// TwinCAT 3 PLC project PLC_Classification
// ProgramVersion: 3.1.4024.0
// libraries:
//   Tc2_Standard, * (Beckhoff Automation GmbH)
//   Tc2_System, * (Beckhoff Automation GmbH)
//   Tc3_Module, * (Beckhoff Automation GmbH)
//   Tc3_Vision, * (Beckhoff Automation GmbH)
// project tree:
//   DUTs/ ST_ClassifierParams.TcDUT, E_ClassifierType.TcDUT, ESvmClassifierType.TcDUT
//   / PlcTask.TcTTO
//   POUs/ FB_TrainingDataHandler.TcPOU, F_ExtractFeatures.TcPOU (not stored), MAIN.TcPOU
// real-time tasks:
//   TASK PlcTask: cycle T#10ms, priority 20, ADS port 350
//   TASK VnTask ImgAcq (TrainingImages): cycle T#10ms, priority 5, ADS port 351
//   TASK VnTask ImgAcq (TestImages): cycle T#10ms, priority 6, ADS port 352

CONFIGURATION PLC_Classification
    RESOURCE PLC ON TwinCAT3
        TASK PlcTask(INTERVAL := T#10ms, PRIORITY := 20);
        PROGRAM MAIN WITH PlcTask : MAIN;
    END_RESOURCE
END_CONFIGURATION

// ---- DUTs/ST_ClassifierParams.TcDUT
TYPE ST_ClassifierParams :
STRUCT
	nKnnK							:	UDINT 							:=	5;
	nRTreesMaxDepth					:	UDINT							:=	5;			// optional Exp parameter
	nRTreesMinSamples				:	UDINT							:=	10;			// optional Exp parameter
	nRTreesActiveVariables			:	UDINT							:=	0;			// optional Exp parameter
	nRTreesMaxIterations			:	UDINT							:=	50;			// optional Exp parameter
	fRTreesEpsilon					:	LREAL							:=	0.1;		// optional Exp parameter
	fStaRho	                        :	LREAL							:=	0.92;
	nStaNu	                        :	UDINT							:=	3;			// optional Exp parameter
	bStaDoublePrecision				:	BOOL							:=	FALSE;		// optional Exp parameter
	fStaBetaSbm						:	LREAL							:=	0.0;		// optional Exp parameter
	nStaPhi							:	UDINT							:=	1;			// optional Exp parameter
	nStaTau							:	UDINT							:=	100;		// optional Exp parameter	
	eSvmType						:	ESvmClassifierType				:=	ESvmClassifierType.C;
	fSvmC							:	LREAL							:=	1;
	fSvmNu							:	LREAL							:=	1;
	eSvmKernelType					:	ETcVnSvmKernelType				:=	ETcVnSvmKernelType.TCVN_SKT_RBF;
	fSvmGamma						:	LREAL							:=	1;
	fSvmCoef0						:	LREAL							:=	1;
	fSvmDegree						:	LREAL							:=	5;
	nSvmMaxIterations				:	UDINT							:=	100000;		// optional Exp parameter
	fSvmEpsilon						:	LREAL							:=	0.00001;	// optional Exp parameter
	eSvmSgdClassifierType			:	ETcVnSvmSgdClassifierType		:=	ETcVnSvmSgdClassifierType.TCVN_SSCT_ASGD; 				// optional Exp parameter
	eSvmSgdClassifierMarginType		:	ETcVnSvmSgdClassifierMarginType	:=	ETcVnSvmSgdClassifierMarginType.TCVN_SSCMT_SOFT_MARGIN; // optional Exp parameter
	fSvmSgdMarginRegularization		:	REAL							:=	0.00001;	// optional Exp parameter
	fSvmSgdInitialStepSize			:	REAL							:=	0.05;		// optional Exp parameter
	fSvmSgdStepDecreasingPower		:	REAL							:=	0.75;		// optional Exp parameter
	nSvmSgdMaxIterations			:	UDINT							:=	100000;		// optional Exp parameter
	fSvmSgdEpsilon					:	LREAL							:=	0.00001;	// optional Exp parameter
END_STRUCT
END_TYPE

// ---- DUTs/E_ClassifierType.TcDUT
{attribute 'qualified_only'}
{attribute 'strict'}
TYPE E_ClassifierType :
(
	KNN := 0,
	NBC,
	RTrees,
	STA,
	SVM,
	SVM_SGD
);
END_TYPE

// ---- DUTs/ESvmClassifierType.TcDUT
{attribute 'qualified_only'}
{attribute 'strict'}
TYPE ESvmClassifierType :
(
	C := TO_UDINT(ETcVnSvm.TCVN_SVM_C_CLASSIFIER),
	NU := TO_UDINT(ETcVnSvm.TCVN_SVM_NU_CLASSIFIER)
) UDINT;
END_TYPE

// ---- POUs/MAIN.TcPOU
PROGRAM MAIN
VAR
	eClassifierType		:	E_ClassifierType;		// Classification type
	stParams			:	ST_ClassifierParams;	// Classification parameters
	bResetModel			:	BOOL;					// Reset model to start a new training with a changed model or parameters
	bResetTrainingData	:	BOOL;					// Reset the trained features to get new ones and train model
	eTrainedModelType	: 	E_ClassifierType;
	
	hrTrain				:	HRESULT;
	hrTest				:	HRESULT;
	
	ipImageTest			:	ITcVnImage;
	ipImageResDisp		:	ITcVnDisplayableImage;
	
	eCameraState		:	ETcVnCameraState;	
	fbCameraTest		:	FB_VN_SimpleCameraControl;
	
	fbTrainingDataHandler:	FB_TrainingDataHandler;
	
	ipClassifierModel	:	ITcVnMlModel;
	ipSamplesTraining	:	ITcVnContainer;
	ipClassLabels		:	ITcVnContainer;
	ipClassLabelsWork	:	ITcVnContainer;
	ipFeatureScaling	:	ITcVnContainer;
	ipSampleTest		:	ITcVnContainer;
	nPredictedClass		:	DINT;
	fNovelty			:	REAL;
	
	// Result
	fNoveltyThreshold	:	REAL;
	sLabel				:	STRING(255);
	aClassNames			:	ARRAY[0..1] OF STRING := ['Apple', 'Banana'];
	aGreen				:	TcVnVector4_LREAL := [0, 255, 0];
END_VAR

// Disclaimer

// This publication contains statements about the suitability of our products for certain
// areas of application. These statements are based on typical features of our products.
// The examples shown in this publication are for demonstration purposes only.
// The information provided herein should not be regarded as specific operation characteristics.
// It is incumbent on the customer to check and decide whether a product is suitable for use
// in a particular application. We do not give any warranty that the source code which is
// made available with this publication is complete or accurate.

// THE SAMPLE CODE CONTAINED IN THIS PUBLICATION IS PROVIDED “AS IS” WITHOUT WARRANTY OF ANY KIND,
// EITHER EXPRESSED, IMPLIED OR STATUTORY, INCLUDING WITHOUT LIMITATION, ANY WARRANTY WITH RESPECT TO NON-INFRINGEMENT,
// FREEDOM FROM PROPRIETARY RIGHTS OF THIRD PARTIES OR FITNESS FOR ANY PARTICULAR PURPOSE.

// This publication may be changed from time to time without prior notice.
// No liability is assumed for errors and/or omissions.
// Our products are described in detail in our data sheets and documentations.
// Product-specific warnings and cautions must be observed.
// For the latest version of our data sheets and documentations visit our website (www.beckhoff.de).

// © Beckhoff Automation GmbH & Co. KG, December 2023

// The reproduction, distribution and utilization of this document as well as the communication
// of its contents to others without express authorization is prohibited. 
// Offenders will be held liable for the payment of damages.
// All rights reserved in the event of the grant of a patent, utility model or design.

//	==========================================================================================

// SAMPLE - Machine Learning Classification
//	-------------------------------------------------------

// Steps To Do:
// ------------
// 1. Add the training images to the TrainingImages control
// 2. Add the test images to the TestingImages control
// 3. Activate the configuration -> Start TwinCAT system and PLC to run -> watch the results in the ADS Image Watch
// 4. Change eClassifierType and stParams to change the model or settings
// 5. Set bResetModel to start create a new model and start training
//    Note: If you change to eClassifierType = STA or from this type to another, a bResetTrainingData is automatically performed due to the different scaling of the training data.
// 6. Set bResetTrainingData to get new training data if images or feature extraction changed

// Reset the trained features to get new ones and train model
IF bResetTrainingData
	OR (eTrainedModelType <> E_ClassifierType.STA AND eClassifierType = E_ClassifierType.STA)
	OR (eTrainedModelType = E_ClassifierType.STA AND eClassifierType <> E_ClassifierType.STA) THEN
	
	bResetTrainingData := FALSE;
	fbTrainingDataHandler.Reset();
	FW_SafeRelease(ADR(ipSamplesTraining));
	FW_SafeRelease(ADR(ipClassLabels));
	FW_SafeRelease(ADR(ipClassLabelsWork));
	FW_SafeRelease(ADR(ipFeatureScaling));
	FW_SafeRelease(ADR(ipClassifierModel));
	eTrainedModelType := eClassifierType;
	// Reset return value
	hrTrain := S_OK;
END_IF

// Get sample data for training
fbTrainingDataHandler(eClassifierType := eClassifierType);
IF ipSamplesTraining = 0 AND ipClassLabels = 0 AND ipFeatureScaling = 0 THEN
	hrTrain := fbTrainingDataHandler.GetTrainingData(ipSamplesTraining, ipClassLabels, ipFeatureScaling);
	hrTrain := F_VN_CopyContainer(ipClassLabels, ipClassLabelsWork, hrTrain);
END_IF

// Retrain with changed model or parameters
IF bResetModel THEN
	bResetModel := FALSE;
	FW_SafeRelease(ADR(ipClassifierModel));
	hrTrain := F_VN_CopyContainer(ipClassLabels, ipClassLabelsWork, hrTrain);
	eTrainedModelType := eClassifierType;
	// Reset return value
	hrTrain := S_OK;
END_IF

IF SUCCEEDED(hrTrain) AND ipSamplesTraining <> 0 AND ipClassLabels <> 0 AND ipClassifierModel = 0 THEN
	
	// Create the model
	CASE eClassifierType OF
		
		E_ClassifierType.KNN:
			hrTrain := F_VN_CreateKnnModel(
								ipMlModel				:=	ipClassifierModel,
								eKnnType				:=	TCVN_KNN_CLASSIFIER,
								nK						:=	stParams.nKnnK,
								hrPrev					:=	hrTrain);
								
			// Set novelty threshold according to model results 
			fNoveltyThreshold := 0.03;
			
		E_ClassifierType.NBC:
			hrTrain := F_VN_CreateNbcModel(
								ipMlModel				:=	ipClassifierModel,
								eNbcType				:=	TCVN_NBC_CLASSIFIER,
								hrPrev					:=	hrTrain);
			
			// Set novelty threshold according to model results
			fNoveltyThreshold := 4.0;
			
		E_ClassifierType.RTrees:
			hrTrain := F_VN_CreateRTreesModelExp(
								ipMlModel				:=	ipClassifierModel,
								eRTreesType				:=	TCVN_RT_CLASSIFIER,
								nMaxDepth				:=	stParams.nRTreesMaxDepth,
								nMinSamples				:=	stParams.nRTreesMinSamples,
								nActiveVariables		:=	stParams.nRTreesActiveVariables,
								nMaxiterations			:=	stParams.nRTreesMaxIterations,
								fEpsilon				:=	stParams.fRTreesEpsilon,
								hrPrev					:=	hrTrain);

		E_ClassifierType.STA:
			hrTrain := F_VN_CreateStaModelExp2(
									ipMlModel           :=	ipClassifierModel,
									eStaType            :=	TCVN_STA_CLASSIFIER,
									fRho                :=	stParams.fStaRho,
									nNu                 :=	stParams.nStaNu,
									bDoublePrecision    :=	stParams.bStaDoublePrecision,
									fBetaSbm			:=	stParams.fStaBetaSbm, 
									nPhi				:=	stParams.nStaPhi, 
									nTau				:=	stParams.nStaTau, 
									hrPrev				:=	hrTrain); 
			
			// Set novelty threshold according to model results
			fNoveltyThreshold := 0.2;
		
		E_ClassifierType.SVM:
			hrTrain := F_VN_CreateSvmModelExp(
								ipMlModel				:=	ipClassifierModel,
								eSvmType				:=	TO_UDINT(stParams.eSvmType),
								fC						:=	stParams.fSvmC,
								fNu						:=	stParams.fSvmNu,
								fP						:=	0,
								eKernelType				:=	stParams.eSvmKernelType,
								fGamma					:=	stParams.fSvmGamma,
								fCoef0					:=	stParams.fSvmCoef0,
								fDegree					:=	stParams.fSvmDegree,
								nMaxIterations			:=	stParams.nSvmMaxIterations,
								fEpsilon				:=	stParams.fSvmEpsilon,
								hrPrev					:=	hrTrain);
			
		E_ClassifierType.SVM_SGD:
			hrTrain := F_VN_CreateSvmSgdClassifierExp(
								ipMlModel				:=	ipClassifierModel,
								eType					:=	stParams.eSvmSgdClassifierType,
								eMarginType				:=	stParams.eSvmSgdClassifierMarginType,
								fMarginRegularization	:=	stParams.fSvmSgdMarginRegularization,
								fInitialStepSize		:=	stParams.fSvmSgdInitialStepSize,
								fStepDecreasingPower	:=	stParams.fSvmSgdStepDecreasingPower,
								nMaxIterations			:=	stParams.nSvmSgdMaxIterations,
								fEpsilon				:=	stParams.fSvmSgdEpsilon,
								hrPrev					:=	hrTrain);
	
			// Change class labels from [0,1] to [-1,1] to be compatilbe with the SvmSgdClassifier model
			hrTrain := F_VN_MultiplyWithContainerElements1(2.0, ipClassLabelsWork, hrTrain);					
			hrTrain := F_VN_AddToContainerElements_DINT(-1, ipClassLabelsWork, hrTrain);
	END_CASE
	
	// Train model
	hrTrain := F_VN_TrainBatch(
					ipMlModel	:=	ipClassifierModel,
					ipSamples	:=	ipSamplesTraining,
					ipOutputs	:=	ipClassLabelsWork,
					hrPrev		:=	hrTrain);

END_IF

// Get test images
eCameraState := fbCameraTest.GetState();

IF eCameraState = TCVN_CS_ERROR THEN
	hrTest := fbCameraTest.Reset();

ELSIF eCameraState < TCVN_CS_ACQUIRING THEN
	hrTest := fbCameraTest.StartAcquisition();

// Camera streaming
ELSIF eCameraState = TCVN_CS_ACQUIRING THEN
	hrTest := fbCameraTest.GetCurrentImage(ipImageTest);

	// Check if new image was received
	IF SUCCEEDED(hrTest) AND ipImageTest <> 0 THEN

        IF ipClassifierModel <> 0 AND ipFeatureScaling <> 0 THEN
			// Get features from sample image and scale 
			hrTest := F_ExtractFeatures(ipImageTest, ipSampleTest, hrTest);
			IF eClassifierType = E_ClassifierType.STA THEN
				hrTest := F_VN_FeatureScalingExp(ipSampleTest, ipFeatureScaling, ipSampleTest, 0.1, 0.9, hrTest);
			ELSE
				hrTest := F_VN_FeatureScaling(ipSampleTest, ipFeatureScaling, ipSampleTest, hrTest);
			END_IF
			
			// Prediction with optional novelty calculation if supported
			CASE eClassifierType OF
				
				E_ClassifierType.KNN, E_ClassifierType.NBC, E_ClassifierType.STA:
					// Predict classification result and novelty
					hrTest := F_VN_PredictSampleClassExp(ipClassifierModel, ipSampleTest, nPredictedClass, fNovelty, hrTest);
				
					// Check the degree of novelty and get result
					IF fNovelty <= fNoveltyThreshold THEN
						sLabel := CONCAT('Prediction: ',aClassNames[nPredictedClass]);
					ELSE
						sLabel := 'Prediction: Unknown';
					END_IF
			ELSE
				// Predict classification result
				hrTest := F_VN_PredictSampleClass(ipClassifierModel, ipSampleTest, nPredictedClass, hrTest);
				
				// Change predicted result for SvmSgdClassifier model and get result
				IF eClassifierType = E_ClassifierType.SVM_SGD AND nPredictedClass < 0 THEN 
					nPredictedClass := nPredictedClass + 1; 
				END_IF
				sLabel := CONCAT('Prediction: ',aClassNames[nPredictedClass]);
			END_CASE
			
			// Write result
			hrTest := F_VN_PutTextExp(sLabel, ipImageTest, 30, 60, TCVN_FT_HERSHEY_PLAIN, 4, aGreen, 2, TCVN_LT_ANTIALIASED, FALSE, hrTest);
		END_IF
		
		// Display Image
		hrTest := F_VN_TransformIntoDisplayableImage(ipImageTest, ipImageResDisp, S_OK);
	END_IF
END_IF

END_PROGRAM

// ---- POUs/FB_TrainingDataHandler.TcPOU
FUNCTION_BLOCK PUBLIC FB_TrainingDataHandler
VAR_INPUT
	eClassifierType		:	E_ClassifierType;
END_VAR
VAR_OUTPUT
END_VAR
VAR
	hr					: HRESULT;
	eCameraState		: ETcVnCameraState;
	fbCameraTraining	: FB_VN_SimpleCameraControl;	
	ipImageTraining		: ITcVnImage;
	ipImageTrainingDisp	: ITcVnDisplayableImage;
	bTrigger			: BOOL := TRUE;
	sLabel				: STRING(255);
	aGreen				: TcVnVector4_LREAL := [0, 255, 0];
	
	// Image Info
	nImagesTotal		: UDINT := 12;
	nImagesLoaded		: UDINT := 0;
	
	ipFeatures			: ITcVnContainer;
	ipImageFeatures		: ITcVnContainer;
	ipLabels			: ITcVnContainer;
	ipScales			: ITcVnContainer;
	ipScaledFeatures	: ITcVnContainer;
END_VAR

// Initialize container
IF ipImageFeatures = 0 THEN
	hr := F_VN_CreateContainer(ipImageFeatures, ContainerType_Vector_Vector_LREAL, nImagesTotal, hr);
	hr := F_VN_CreateContainer(ipLabels, ContainerType_Vector_DINT, nImagesTotal, hr);
END_IF

// Get training images
eCameraState := fbCameraTraining.GetState();

IF eCameraState = TCVN_CS_ERROR THEN
	hr := fbCameraTraining.Reset();
	
// Camera trigger image
ELSIF eCameraState = TCVN_CS_TRIGGERING THEN
	hr := fbCameraTraining.TriggerImage();
	
ELSIF eCameraState < TCVN_CS_ACQUIRING THEN
	hr := fbCameraTraining.StartAcquisition();

// Camera streaming
ELSIF eCameraState = TCVN_CS_ACQUIRING THEN

	IF bTrigger THEN
		hr := fbCameraTraining.TriggerImage();
		IF SUCCEEDED(hr) THEN
			bTrigger := FALSE;
		END_IF
	ELSE
		hr := fbCameraTraining.GetCurrentImage(ipImageTraining);

		// Check if new image was received
		IF SUCCEEDED(hr) AND ipImageTraining <> 0 THEN
			
			// Get features from training image 
			hr := F_ExtractFeatures(ipImageTraining, ipFeatures, hr);
		
			// Add features and label to the containers. First class label = 0, second class = 1
			hr := F_VN_SetAt_ITcVnContainer(ipFeatures, ipImageFeatures, nImagesLoaded, hr);
			FW_SafeRelease(ADR(ipFeatures));
			hr := F_VN_SetAt_DINT(UDINT_TO_DINT(nImagesLoaded / 6), ipLabels, nImagesLoaded, hr);
			
			// Display image
			sLabel := CONCAT('Image Number: ', UDINT_TO_STRING(nImagesLoaded + 1));
			hr := F_VN_PutTextExp(sLabel, ipImageTraining, 30, 60, TCVN_FT_HERSHEY_PLAIN, 4, aGreen, 2, TCVN_LT_ANTIALIASED, FALSE, hr);
			hr := F_VN_TransformIntoDisplayableImage(ipImageTraining, ipImageTrainingDisp, hr);
			
			nImagesLoaded := nImagesLoaded + 1;
			IF nImagesLoaded < nImagesTotal THEN
				// Trigger next image
				bTrigger := TRUE;
			ELSE
				// After collecting all training data, normalize the feature values
				hr := F_VN_GetFeatureScales(ipImageFeatures, ipScales, TCVN_FST1_MINMAX, hr);
				IF eClassifierType = E_ClassifierType.STA THEN
					hr := F_VN_FeatureScalingExp(ipImageFeatures, ipScales, ipScaledFeatures, 0.1, 0.9, hr);
				ELSE
					hr := F_VN_FeatureScaling(ipImageFeatures, ipScales, ipScaledFeatures, hr);
				END_IF
				FW_SafeRelease(ADR(ipImageFeatures));
			END_IF
		END_IF
	END_IF
END_IF

METHOD PUBLIC GetTrainingData : HRESULT
VAR_INPUT
	ipTrainingSamples	: REFERENCE TO ITcVnContainer;
	ipClassLabels		: REFERENCE TO ITcVnContainer;
	ipFeatureScaling	: REFERENCE TO ITcVnContainer;
END_VAR
VAR
	hr					: HRESULT;
END_VAR
IF nImagesLoaded = nImagesTotal THEN
	hr := F_VN_CopyContainer(ipScaledFeatures, ipTrainingSamples, hr);
	hr := F_VN_CopyContainer(ipLabels, ipClassLabels, hr);
	GetTrainingData := F_VN_CopyContainer(ipScales, ipFeatureScaling, hr);
ELSE
	GetTrainingData := S_PENDING;
END_IF
END_METHOD

METHOD PUBLIC Reset : HRESULT
VAR_INPUT
END_VAR
nImagesLoaded := 0;
FW_SafeRelease(ADR(ipFeatures));
FW_SafeRelease(ADR(ipImageFeatures));
FW_SafeRelease(ADR(ipLabels));
FW_SafeRelease(ADR(ipScales));
FW_SafeRelease(ADR(ipScaledFeatures));
bTrigger := TRUE;
END_METHOD

END_FUNCTION_BLOCK
